// TwinCAT 3 PLC project MainPlc
// ProgramVersion: 3.1.4024.0
// libraries:
//   Tc2_Standard, * (Beckhoff Automation GmbH)
//   Tc2_System, * (Beckhoff Automation GmbH)
//   Tc3_Module, * (Beckhoff Automation GmbH)
// project tree:
//   / PlcTask.TcTTO
//   POUs/ MAIN.TcPOU
// real-time tasks:
//   TASK PlcTask: cycle T#10ms, priority 6, ADS port 350

CONFIGURATION MainPlc
    RESOURCE PLC ON TwinCAT3
        TASK PlcTask(INTERVAL := T#10ms, PRIORITY := 6);
        PROGRAM MAIN WITH PlcTask : MAIN;
    END_RESOURCE
END_CONFIGURATION

// ---- POUs/MAIN.TcPOU
PROGRAM MAIN
VAR
	runOnlyOnce : BOOL := FALSE;
END_VAR

IF NOT runOnlyOnce THEN
ADSLOGSTR(msgCtrlMask := ADSLOG_MSGTYPE_ERROR OR ADSLOG_MSGTYPE_LOG, msgFmtStr := 'Hello World',strArg := '');
	runOnlyOnce := TRUE;
	END_IF

END_PROGRAM
